FUNCTION_BLOCK ConveyorController
  (* Standard: 61499-2 *)
  (* Version 0.1, 2016-00-28, hpea485, UOA *)
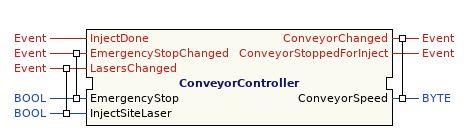
  EVENT_INPUT
    InjectDone;
    EmergencyStopChanged WITH EmergencyStop;
    LasersChanged WITH InjectSiteLaser;
  END_EVENT
  EVENT_OUTPUT
    ConveyorChanged WITH ConveyorSpeed;
    ConveyorStoppedForInject;
  END_EVENT
  VAR_INPUT
    EmergencyStop : BOOL;
    InjectSiteLaser : BOOL;
  END_VAR
  VAR_OUTPUT
    ConveyorSpeed : BYTE;
  END_VAR
  VAR
    Variable1 : BOOL;
  END_VAR
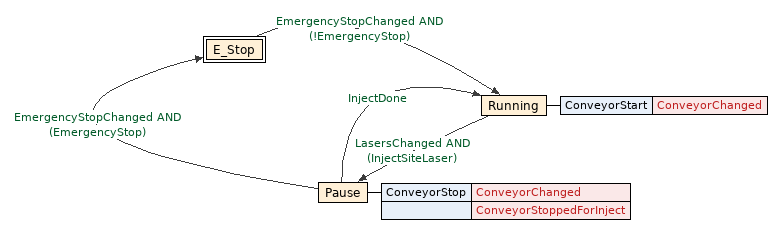
  EC_STATES
    E_Stop;
    Running : ConveyorStart -> ConveyorChanged;
    Pause : ConveyorStop -> ConveyorChanged, -> ConveyorStoppedForInject;
  END_STATES
  EC_TRANSITIONS
    Pause TO Running := InjectDone;
    Pause TO E_Stop := EmergencyStopChanged AND (EmergencyStop);
    Running TO Pause := LasersChanged AND (InjectSiteLaser);
    E_Stop TO Running := EmergencyStopChanged AND (!EmergencyStop);
  END_TRANSITIONS
  ALGORITHM ConveyorStart IN VHDL:
ConveyorSpeed <= 1;
  END_ALGORITHM
  ALGORITHM ConveyorStop IN VHDL:
ConveyorSpeed <= 0;
  END_ALGORITHM
  ALGORITHM ConveyorRunning IN VHDL:

  END_ALGORITHM
  ALGORITHM ConveyorEStop IN VHDL:

  END_ALGORITHM
END_FUNCTION_BLOCK
